FUNCTION_BLOCK FB_RecipeFactory
VAR
    BuilderWings : FB_RecipeBuilderWings;
    BuilderFlaps : FB_RecipeBuilderFlaps;
    BuilderArona : FB_RecipeBuilderArona;
END_VAR

METHOD GetBuilder : I_RecipeBuilder
VAR_INPUT
    RequestedRecipe : E_RecipeID;
END_VAR
CASE RequestedRecipe OF
    E_RecipeID.eBorgoWings:
        GetBuilder := BuilderWings; 
        
    E_RecipeID.eBorgoFlaps:
        GetBuilder := BuilderFlaps;
        
    E_RecipeID.eArona:
        GetBuilder := BuilderArona;
        
ELSE
    // Jeśli ktoś poda złe ID, zwracamy "nic" (0)
    GetBuilder := 0; 
END_CASE
END_METHOD

METHOD InitializeFactory
VAR_INPUT
    Config : ST_RecipeBuilder_Config;
END_VAR
BuilderWings.Config := Config;
BuilderFlaps.Config := Config;
BuilderArona.Config := Config;
END_METHOD

METHOD UpdateConfig
VAR_INPUT
    Config : ST_RecipeBuilder_Config;
END_VAR
// Fabryka rozsyła nową konfigurację do wszystkich swoich "dzieci"
BuilderWings.Config := Config;
BuilderFlaps.Config := Config;
BuilderArona.Config := Config;
END_METHOD

END_FUNCTION_BLOCK

(* stored: Version 1.1.0.1, ProductVersion 3.1.4024.15
   POU FB_RecipeFactory: Id {eb67f754-8d88-44c2-acf6-733dd105dd46}, SpecialFunc None
   Method GetBuilder: Id {4ef94639-3187-4b95-bdcd-c7a9da21c9f0}
   Method InitializeFactory: Id {d617016c-6308-411a-9cc3-c9f77798a181}
   Method UpdateConfig: Id {addb126c-7b31-4fe1-bab5-a92c30ad08f7} *)
